S      V300.1, 1                   // M_Alarm_Overflow_BHighR      Q0.4, 1                     // 关阀CMOVW   99, VW2MOVB   2, VB270                    // 故障JMP    6
// 诊断子状态调度LDW=   VW264, 0JMP    1LDW=   VW264, 1JMP    2LDW=   VW264, 2JMP    3LDW=   VW264, 3JMP    4LDW=   VW264, 4JMP    5JMP    6
// ---- 子状态0: 空闲 ----// S0空闲LBL    1JMP    6
// ---- 子状态1: 等待开到位 ----// S1等待开到位LBL    2// T56开到位超时 + T57排水超时(两套独立判据, PT均=VW276)LD     SM0.0TON    T56, VW276                  // PT=VD_Timeout_ValveC(VD54)×10TON    T57, VW276                  // 排水超时: 液位低位未在VD_Timeout_ValveC内到达
// 开到位=ON → 转S2排水中// [已修复 v2.2] 用 V63.2 缓存 EU 结果,避免 R 指令链栈空LD     I8.4EU=      V63.2LD     V63.2MOVW   2, VW264LD     V63.2R      T56, 1LD     V63.2R      T57, 1JMP    6
// 开到位超时 → 报警46LD     T56S      V302.6, 1                   // M_Alarm_ValveC_OpenTimeoutMOVW   99, VW2MOVW   2, VW270JMP    6
// 排水超时(开阀后液位低位仍未到达) → 报警60LD     T57AN     I1.0                        // 确认液位计B低位仍OFFS      V303.0, 1                   // M_Alarm_ValveC_CloseTimeout(排水超时同用码60)MOVW   99, VW2MOVW   2, VW270JMP    6
// ---- 子状态2: 排水中(等待液位低位) ----// S2排水中LBL    3// 液位计B低位=ON → 转S3延时验证LD     I1.0MOVW   3, VW264JMP    6// 液位低位=OFF → 继续排水,无动作
// ---- 子状态3: 延时验证(液位低位须持续ON) ----// S3延时验证LBL    4// I1.0持续ON达VD_Delay_ValveC_Verify → 排水完成,关阀C// 注: I1.0中途OFF时TON输入断开,T101自动清零,液位低位须连续保持LD     I1.0TON    T101, VW284                  // PT=VD_Delay_ValveC_Verify(VD472)×10LD     T101R      Q0.4, 1                     // 关阀CMOVW   4, VW264                    // 转S4等关到位JMP    6// 液位低位丢失 → 回S2排水中(T101已自动复位)LDN    I1.0MOVW   2, VW264JMP    6
// ---- 子状态4: 等待关到位 ----// S4等待关到位LBL    5// T58关到位超时LD     SM0.0TON    T58, VW276                  // PT=VD_Timeout_ValveC×10
// 关到位=ON → 正常完成// [已修复 v2.2] 用 V63.3 缓存条件,避免 R 指令链栈空LD     I8.5=      V63.3LD     V63.3MOVW   0, VW264                    // VW264=0空闲LD     V63.3MOVW   1, VW270                    // Diag_Result_C=1正常完成LD     V63.3R      T58, 1JMP    6
// 关到位超时 → 报警60LD     T58AN     I8.5S      V303.0, 1                   // M_Alarm_ValveC_CloseTimeoutMOVW   99, VW2MOVW   2, VW270                    // Diag_Result_C=2故障(已修正:用MOVW)JMP    6
// 诊断结束LBL    6

// ============================================================// 文件结束// 说明://   1. FC17调用本FC前置VW264=1启动//   2. FC17检查VW270: 0等待, 1正常完成转S5/S7, 2故障//   3. VW276=VD_Timeout_ValveC(VD54)×10转换值//      VW284=VD_Delay_ValveC_Verify(VD472)×10转换值【v10.4新增】//   4. 【v10.4硬件变更】I0.2保留未使用//      V302.5/V302.7/V303.1改为保留位(报警码45/47/61废弃,不再置位)//      T57由"流量开关超时"改制为"排水超时"(液位低位到达超时)//      排水异常=开到位超时(46)或排水/关到位超时(60)//   5. VW270写入统一用MOVW(写完整WORD),确保FC17的AW=VW270判断正确// ============================================================

JMP    6
LBL    1
JMP    6
LBL    2
LD     SM0.0
TON    T56, VW276
TON    T57, VW276
LD     I8.4
EU
=      V63.2
LD     V63.2
MOVW   2, VW264
LD     V63.2
R      T56, 1
LD     V63.2
R      T57, 1
JMP    6
LD     T56
S      V302.6, 1
MOVW   99, VW2
MOVW   2, VW270
JMP    6
LD     T57
AN     I1.0
S      V303.0, 1
MOVW   99, VW2
MOVW   2, VW270
JMP    6
LBL    3
LD     I1.0
MOVW   3, VW264
JMP    6
LBL    4
LD     I1.0
TON    T101, VW284
LD     T101
R      Q0.4, 1
MOVW   4, VW264
JMP    6
LDN    I1.0
MOVW   2, VW264
JMP    6
LBL    5
LD     SM0.0
TON    T58, VW276
LD     I8.5
=      V63.3
LD     V63.3
MOVW   0, VW264
LD     V63.3
MOVW   1, VW270
LD     V63.3
R      T58, 1
JMP    6
LD     T58
AN     I8.5
S      V303.0, 1
MOVW   99, VW2
MOVW   2, VW270
JMP    6
LBL    6
END_SUBROUTINE_BLOCK
SUBROUTINE_BLOCK RhythmCorrection:SBR19
TITLE=// ============================================================
// // 文件: FC40_RhythmCorrection.stl
// // 功能: 双倒计时器周期管理(v2.2 重写,替代原三层纠偏)
// // Story: v2.2 流程重构 (替代 AQEX-8 节奏纠偏)
// // 说明: v2.2 取消原"三层自动纠偏"机制,改为通过 FC40 管理两个交替工作
// //       的 32 位秒计数器(VD248/VD252),严格保证 24h 换水次数硬约束
// // 调用: OB1 每周期调用(在 FC1 状态调度之前)
// // 输出: 触发 S6 排水 / 触发下一轮 S1 / 倒计时到 0 报警 / 双计时器显示值
// // ============================================================
//
// // 符号说明:
// // VD414 : VD_24h_Target           24h 换水目标次数 (HMI 设定)
// // VD426 : VD_Transfer_Margin      周期尾端转移余量 (秒, 默认 30, HMI 设定)
// // VD430 : VD_Prep_Safety_Margin   上缸配液安全余量 (秒, 默认 10, HMI 设定)
// // VD186 : VD_T_cycle              本轮倒计时总时长(秒,内部中间变量)
// // VD248 : VD_TimerA_Elapsed       TimerA 已运行秒数(32 位 REAL)
// // VD252 : VD_TimerB_Elapsed       TimerB 已运行秒数(32 位 REAL)
// // VD256 : VD_TimerA_Display       TimerA 显示值(秒, DINT, HMI 读取)
// // VD244 : VD_TimerB_Display       TimerB 显示值(秒, DINT, HMI 读取)
// // T63   : T_1s_Pulse              1 秒脉冲发生器(100ms 时基,PT=10)
// // V63.4 : M_1s_Pulse              1 秒脉冲 EU 缓存
// // V63.5 : M_S6Trig_Cache          S6触发条件缓存(v2.3, 避免LPS/LPP/ALD栈消耗)
// // V63.6 : M_NextS1Trig_Cache      下一轮S1触发条件缓存(v2.3)
// // V63.7 : M_CycleTimeout_Cache    周期超时报警条件缓存(v2.3)
// // AC2   : 运算中间值(v2.3 NET5 T_cycle-Prep_Needed 阈值)
// // VW2   : 下缸主状态机
// // VW418 : 上缸配液子流程状态
// // VW6   : 当前报警码 (=0 才允许触发)
// // VW400 : 已完成换水次数 (v2.3.2由VW306迁入, 避让手动命令位V306.0~V307.3)
// // VD70  : S1 实测时长 (秒)
// // VD28  : S2 搅拌固定时长 (秒)
// // VD116 : S6 滚动实测时长 (秒,首轮为S4实测值)
// // M16.0 : M_TimerA_Active         当前下缸轮次使用 TimerA 标志
// // M16.1 : M_NextCycleTrigger      触发下一轮 S1 脉冲
// // V303.6: M_Alarm_CycleTimeout    单轮换水周期超时报警
BEGIN
Network 1
//  计算 T_single 和 T_cycle
//  T_single = 86400.0 / VD414          // 单次目标周期(秒)
//  T_cycle = T_single - VD426 - VD430  // 实际倒计时总时长(秒)
LD     SM0.0MOVR   86400.0, VD186/R     VD414, VD186                 // T_single-R     VD426, VD186                 // - Transfer_Margin-R     VD430, VD186                 // - Safety_Margin = T_cycle

// T_cycle <= 0 检查:周期参数过激进,报警并禁止启动LD     SM0.0AR>    VD186, 0.0                   // T_cycle > 0 ?JMP    10                          // 是 → 正常路径// 否 → 参数过激进LD     SM0.0S      V303.6, 1                   // M_Alarm_CycleTimeout=1(强制人工确认)JMP    9                           // → 跳到本FC末尾
LBL    10// 正常路径继续JMP    10
LD     SM0.0
S      V303.6, 1
JMP    9
LBL    10
Network 2
//  1 秒脉冲发生器(100ms 时基,PT=10)
//  [已修复 v2.2] 用 T63 产生 1s 脉冲,驱动 32 位秒计数器,不受 32767 限制
LD     SM0.0R      T63, 1TON    T63, 10LD     T63EU=      V63.4                       // 1 秒脉冲 EU 缓存R      T63, 1
TON    T63, 10
LD     T63
EU
=      V63.4
Network 3
//  双倒计时器累加:本轮进行中,每秒给当前活动计时器 +1
//  【v2.3修复】原门控"仅VW418=1(S1期间)"导致Elapsed只计到S1结束,
//    NET4/NET5的T_cycle比较式永远无法触发;改为"本轮进行中"门控:
//    VW418≠0(上缸子流程进行中) 且 VW2?{0,7,8,99}(非S0/S6/S7/S_ERROR)
//    计时区间为 本轮S6完成→本轮S6触发(排水窗口冻结,与NET4阈值语义对齐)
//  【2026-09-25修复】增加 VW2≠7: S6排水期间冻结计数,消除排水末越界误报
LD     V63.4                       // 1 秒脉冲LDW<>  VW418, 0                    // 上缸子流程进行中(1/2/3/4)AW<>   VW2, 0                      // 非S0AW<>   VW2, 7                      // 【2026-09-25修复】非S6(排水窗口冻结计数,消除越界误报)AW<>   VW2, 8                      // 非S7AW<>   VW2, 99                     // 非S_ERRORA      M16.0                       // TimerA 活动?+R     1.0, VD248                  // TimerA_Elapsed + 1LD     V63.4                       // 1 秒脉冲LDW<>  VW418, 0                    // 上缸子流程进行中AW<>   VW2, 0                      // 非S0AW<>   VW2, 7                      // 【2026-09-25修复】非S6(排水窗口冻结计数)AW<>   VW2, 8                      // 非S7AW<>   VW2, 99                     // 非S_ERRORAN     M16.0                       // TimerB 活动?+R     1.0, VD252                  // TimerB_Elapsed + 1Network 4
//  S6 触发条件
//  【v2.3修复】原实现"Elapsed <= VD116"比较方向与语义相反(且代码注释与指令矛盾),
//    按设计语义改为: 本轮剩余 <= S6_actual ? Elapsed >= T_cycle - VD116
//  S6_actual 统一使用 VD116:首轮为S4实测值(由FC15写入),后续为S6滚动实测值(由FC17写入)
LD     SM0.0LPSA      M16.0                       // 当前 TimerA?MOVR   VD248, AC0                  // AC0 = TimerA_ElapsedLPPLPSAN     M16.0                       // 当前 TimerB?MOVR   VD252, AC0                  // AC0 = TimerB_ElapsedLPPOLD                                // 选择当前活动 ElapsedMOVR   VD186, AC1                  // AC1 = T_cycle-R     VD116, AC1                  // AC1 = T_cycle - S6_actual (S6触发阈值)-R     AC1, AC0                    // AC0 = Elapsed - 阈值AR>=   AC0, 0.0                    // Elapsed >= T_cycle - S6_actual ?AW=    VW2, 6                      // 当前在 S5AW=    VW6, 0                      // 无报警=      V63.5                       // 缓存S6触发条件(避免LPS/LPP/ALD栈消耗丢弃门控)LD     V63.5MOVW   7, VW2                      // 转 S6 排水LD     V63.5S      M10.7, 1                    // 【v2.3修复】置S6首次进入脉冲(原FC16已删除置位,FC17无源可取)AW=    VW2, 6
AW=    VW6, 0
=      V63.5
LD     V63.5
MOVW   7, VW2
LD     V63.5
S      M10.7, 1
Network 5
//  下一轮 S1 触发条件
//  【v2.3修复】原实现"Elapsed >= Prep_Needed"漏T_cycle项,且要求VW418=0(死条件);
//    按设计语义改为: 本轮剩余 <= Prep_Needed ? Elapsed >= T_cycle - Prep_Needed,
//    门控改为 VW418=4(上缸已转移,可启动下一轮配液)
//  Prep_Needed = VD70 + VD28 + VD430 (S1 实测 + S2 固定 + 上缸安全余量)
LD     SM0.0LPSA      M16.0                       // 当前 TimerA?MOVR   VD248, AC0                  // AC0 = TimerA_ElapsedLPPLPSAN     M16.0                       // 当前 TimerB?MOVR   VD252, AC0                  // AC0 = TimerB_ElapsedLPPOLD                                // 选择当前活动 ElapsedMOVR   VD70, AC1                   // AC1 = S1_Actual+R     VD28, AC1                   // + S2 固定+R     VD430, AC1                  // + 安全余量 = Prep_NeededMOVR   VD186, AC2                  // AC2 = T_cycle-R     AC1, AC2                    // AC2 = T_cycle - Prep_Needed (下一轮S1触发阈值)-R     AC2, AC0                    // AC0 = Elapsed - 阈值AR>=   AC0, 0.0                    // Elapsed >= T_cycle - Prep_Needed ?AW=    VW418, 4                    // 【v2.3修复】上缸已转移(原VW418=0为死状态)AW=    VW6, 0                      // 无报警=      V63.6                       // 缓存触发条件LD     V63.6S      M16.1, 1                    // 触发下一轮 S1 脉冲(由OB1消费: VW418 4→1)AR>=   AC0, 0.0
AW=    VW418, 4
AW=    VW6, 0
=      V63.6
LD     V63.6
S      M16.1, 1
Network 6
//  倒计时到 0 报警 (V303.6)
//  报警语义: "错过S6触发窗口"才报 —— Elapsed >= T_cycle 且 NET4 本扫描未触发 S6
//  【2026-09-25修复】原门控仅"不在S7",导致:
//    (a) VD116=0(首轮)时 NET4/NET6 同阈值,NET4先置VW2=7,NET6同扫描误报;
//    (b) S6排水期间 NET3 继续累加,排水末 Elapsed 必然越界,每轮末必报
//    修复: AN V63.5(S6触发缓存) + 排除 VW2=7(S6排水窗口,计数已冻结)
//  【v2.3修复】原LPS/LPP/ALD结构会丢弃门控,改用V位缓存
LD     SM0.0LPSA      M16.0                       // 当前 TimerA?MOVR   VD248, AC0                  // AC0 = TimerA_ElapsedLPPLPSAN     M16.0                       // 当前 TimerB?MOVR   VD252, AC0                  // AC0 = TimerB_ElapsedLPPOLD                                // 选择当前活动 Elapsed-R     VD186, AC0                  // AC0 = Elapsed - T_cycleAR>=   AC0, 0.0                    // Elapsed >= T_cycle ?AN     V63.5                       // 【2026-09-25】NET4未在本扫描触发S6(错过窗口才报)AW<>   VW2, 7                      // 【2026-09-25】不在S6排水窗口(计数冻结,Elapsed不再增长)AW<>   VW2, 8                      // 不在 S7=      V63.7                       // 缓存报警条件LD     V63.7S      V303.6, 1                   // 单轮换水周期超时报警AN     V63.5
AW<>   VW2, 7
AW<>   VW2, 8
=      V63.7
LD     V63.7
S      V303.6, 1
Network 7
//  双倒计时器显示值写入 (HMI 读取)
//  [已修复 v2.2] VD256/VD244 直接显示 Elapsed 秒数(DINT)
LD     M16.0                       // 当前使用 TimerA?
ROUND  VD248, VD256                // VD_TimerA_Display = TimerA_Elapsed (秒)LDN    M16.0                       // 当前使用 TimerB?ROUND  VD252, VD244                // VD_TimerB_Display = TimerB_Elapsed (秒)

LBL    9// 本FC结束// 返回 OB1 (OB1 在调度 FC1 之前调用本FC,保证 M16.1 下一轮 S1 触发脉冲及时响应)

// ============================================================// 文件结束// ============================================================// 说明://   1. 调用时机: OB1 在 FC22(RTC Sync) 之后、FC1(状态调度) 之前调用//   2. 计数器清零: FC11 在 S1 首次进入时清零【非活动】计数器//      (S1启动于本轮中段,活动计数器属于本轮,不能清;计时区间为 S6完成→S6触发)//   3. 计时器切换: S6 完成后由 FC17 切 M16.0 = NOT M16.0(全程序唯一切换点)//   4. 报警 V303.6: 不受 V200.0 模式影响,必须 V0.3 人工确认;//      置位条件为"错过S6触发窗口"(NET4未触发且Elapsed>=T_cycle且不在S6/S7);//      复位由 FC3 NETWORK 4 (V0.3上升沿) 执行: 清V303.6 + 清零VD248/VD252(本轮重新计时),//      FC3A 公共复位不含此位(2026-09-25补漏); 不清计时器则确认后同扫描被NET6重报(死锁)//   5. T_cycle <= 0: 直接报警并跳过本周期其他计算(跳到 LBL 9)//   6. 显示值 VD256/VD244: 真空闲区(原 VD442/VD446 与 VD440/444 字节重叠已迁移)// ============================================================

LBL    9
END_SUBROUTINE_BLOCK
SUBROUTINE_BLOCK MBUS_CTRL:SBR20
TITLE=This code is property of Siemens Industry, Inc.
VAR_INPUT
Mode:BOOL;	//  1 = Modbus, 0 = PPI (stop Modbus)
Baud:DWORD;	//  1200, 2400 ... 115200
Parity:BYTE;	//  0 = none, 1 = odd, 2 = even
Port:BYTE;	// 0 or 1
Timeout:INT;	//  slave response timeout in milliseconds
END_VAR
VAR_OUTPUT
Done:BOOL;	//  Done flag (always set)
Error:BYTE;	//  Error status
END_VAR
VAR
AC0save:DWORD;
AC1save:DWORD;
AC2save:DWORD;
AC3save:DWORD;
END_VAR
BEGIN
Network 1 // 此 POU 针对编辑和查看设置了密码保护.

END_SUBROUTINE_BLOCK
SUBROUTINE_BLOCK MBUS_MSG:SBR21
TITLE=This code is property of Siemens Industry, Inc.
VAR_INPUT
First:BOOL;	// New message (Set to a 1 for only one scan for a new request)
Slave:BYTE;	// Slave address (0 - 247)
RW:BYTE;	// Read = 0, Write = 1
Addr:DWORD;	// Modbus addr (ie 40001)
Count:INT;	// Number of elements (1- 120 words or 1 to 1920 bits)
DataPtr:DWORD;	// Pointer to data (ie &VB100)
END_VAR
VAR_OUTPUT
Done:BOOL;	// Done flag (0 = busy, 1 = done)
Error:BYTE;	// Error (0 = no error)
END_VAR
VAR
AC0save:DWORD;
AC1save:DWORD;
AC2save:DWORD;
END_VAR
BEGIN
Network 1 // 此 POU 针对编辑和查看设置了密码保护.

END_SUBROUTINE_BLOCK
SUBROUTINE_BLOCK MBUSM1:SBR22
TITLE=This code is property of Siemens Industry, Inc.
VAR_OUTPUT
crc:WORD;
END_VAR
VAR
count:INT;
ptr:DWORD;
END_VAR
BEGIN
Network 1 // 此 POU 针对编辑和查看设置了密码保护.

END_SUBROUTINE_BLOCK
SUBROUTINE_BLOCK ManualSyringePump:SBR23
TITLE=
BEGIN
Network 1
//  孤儿态自恢复
//  [已修复 v2.2] 用 V62.2 缓存条件,避免 R 指令链栈空
LDW<>  VW390, 0
AW<>   VW390, 30
AN     M11.6
AN     M11.7
AN     M12.0
AN     M13.5
AN     M13.6
=      V62.2
LD     V62.2
MOVW   0, VW390
LD     V62.2
R      M13.7, 1


// 启动命令检测 - 仅空闲态(VW390=0)响应
// [已修复 v2.2] 用 V62.3 缓存 EU 结果,避免 S/R 指令链栈空
LD     SM0.0
A      V307.2
EU
AW=    VW390, 0
=      V62.3
LD     V62.3
MOVR   0.0, VD392
LD     V62.3
MOVR   VD452, VD396
LD     V62.3
R      M13.7, 1
LD     V62.3
R      M13.5, 1
LD     V62.3
R      M13.6, 1
LD     V62.3
R      M12.0, 1
LD     V62.3
R      M11.6, 1
LD     V62.3
R      M11.7, 1
LD     V62.3
MOVW   1, VW390
LD     V62.3
R      V307.2, 1


// 停止命令检测 - 非空闲态响应
// [已修复 v2.2] 用 V62.4 缓存 EU 结果,避免 S/R 指令链栈空
LD     SM0.0
A      V307.3
EU
AW<>   VW390, 0
=      V62.4
LD     V62.4
S      M13.7, 1
LD     V62.4
R      V307.3, 1


// 全局错误检测
// [已修复 v2.2] 用 V62.5 缓存全局错误条件,避免 R 指令链栈空
LDW=   VW390, 1
OW=    VW390, 2
OW=    VW390, 3
LD     V303.4
LD     SM0.0
AW>=   VW4, 4
OLD
ALD
=      V62.5
LD     V62.5
MOVW   99, VW390
LD     V62.5
R      M13.5, 1
LD     V62.5
R      M13.6, 1
LD     V62.5
R      M13.7, 1
LD     V62.5
R      M12.0, 1
LD     V62.5
R      M11.6, 1
LD     V62.5
R      M11.7, 1


// 子状态1-1 - 计算本次抽液步数
LD     SM0.0
AW=    VW390, 1
AN     M13.5
AN     M11.6
AN     M11.7
AN     M12.0
MOVR   VD396, VD102
/R     VD350, VD102
AR>=   VD102, 6000.0
JMP    10
ROUND  VD102, AC0
MOVR   AC0, VD102
JMP    11
LBL    10
MOVR   6000.0, VD102
LBL    11


// 子状态1-2 - 检查步数并下发抽液指令(40006)
LD     SM0.0
AW=    VW390, 1
AN     M13.5
AN     M11.6
AN     M11.7
AN     M12.0
AW=    VW4, 0
=      V60.4
LD     V60.4
ROUND  VD102, AC0
AR>    AC0, 0.0
JMP    12
// [已修复 v2.2] 复用 V60.4 缓存条件,补齐 R/S 链前面的 LD
LD     V60.4
R      M12.0, 1
LD     V60.4
R      M11.6, 1
LD     V60.4
R      M11.7, 1
LD     V60.4
MOVW   3, VW390
JMP    13
LBL    12
MOVW   AC0, VW204
MOVW   AC0, VW230
MOVD   16#9C46, VD232
LD     V60.4
S      M11.6, 1
LD     V60.4
S      M13.5, 1
LBL    13


// 子状态1-3 - 抽液写失败处理
// [已修复 v2.2] 用 V64.0 缓存条件,避免 S/R 链栈空
LD     M12.0
AW=    VW390, 1
A      V303.4
=      V64.0
LD     V64.0
MOVW   99, VW390
LD     V64.0
R      M13.5, 1
LD     V64.0
R      M13.7, 1
LD     V64.0
R      M12.0, 1
LD     V64.0
R      M11.6, 1
LD     V64.0
R      M11.7, 1


// 子状态1-3 - 抽液写成功处理
// [已修复 v2.2] 用 V64.1 缓存条件,避免 S/R 链栈空
LD     M12.0
AW=    VW390, 1
AN     V303.4
=      V64.1
LD     V64.1
R      M12.0, 1
LD     V64.1
R      M11.6, 1


// 子状态1-4 - 等待抽液执行完成
// [已修复 v2.2] 用 V65.4 缓存条件,避免 R 指令链栈空
LD     M13.5
AW=    VW390, 1
AW=    VW4, 0
AN     M11.6
AN     M11.7
AN     M12.0
=      V65.4
LD     V65.4
R      M13.5, 1
LD     V65.4
MOVW   2, VW390


// 子状态2-1 - 下发排液指令(40007)
// [已修复 v2.2] 用 V65.3 缓存条件,避免 S 指令链栈空
LD     SM0.0
AW=    VW390, 2
AN     M13.6
AN     M11.6
AN     M11.7
AN     M12.0
AW=    VW4, 0
=      V65.3
LD     V65.3
ROUND  VD102, AC0
MOVW   AC0, VW230
MOVW   AC0, VW206
MOVD   16#9C47, VD232
LD     V65.3
S      M11.6, 1
LD     V65.3
S      M13.6, 1


// 子状态2-2 - 排液写失败处理
// [已修复 v2.2] 用 V64.2 缓存条件,避免 S/R 链栈空
LD     M12.0
AW=    VW390, 2
A      V303.4
=      V64.2
LD     V64.2
MOVW   99, VW390
LD     V64.2
R      M13.6, 1
LD     V64.2
R      M13.7, 1
LD     V64.2
R      M12.0, 1
LD     V64.2
R      M11.6, 1
LD     V64.2
R      M11.7, 1


// 子状态2-2 - 排液写成功处理
// [已修复 v2.2] 用 V64.3 缓存条件,避免 S/R 链栈空
LD     M12.0
AW=    VW390, 2
AN     V303.4
=      V64.3
LD     V64.3
R      M12.0, 1
LD     V64.3
R      M11.6, 1


// 子状态2-3 - 等待排液执行完成,累加本循环体积
// [已修复 v2.2] 用 V64.4 缓存条件,避免 S/R 链栈空
LD     M13.6
AW=    VW390, 2
AW=    VW4, 0
AN     M11.6
AN     M11.7
AN     M12.0
=      V64.4
LD     V64.4
MOVR   VD102, AC0
LD     V64.4
*R     VD350, AC0
LD     V64.4
+R     AC0, VD392
LD     V64.4
-R     AC0, VD396
LD     V64.4
R      M13.6, 1


// 子状态2-4 - 判断分支: 停止请求 → 回零
// [已修复 v2.2] 用 V64.5 缓存条件,避免 S/R 链栈空
LD     SM0.0
AW=    VW390, 2
AN     M13.6
A      M13.7
=      V64.5
LD     V64.5
R      M12.0, 1
LD     V64.5
R      M11.6, 1
LD     V64.5
R      M11.7, 1
LD     V64.5
MOVW   3, VW390


// 子状态2-4 - 判断分支: 单次模式 → 回零
// [已修复 v2.2] 用 V64.6 缓存条件,避免 S/R 链栈空
LD     SM0.0
AW=    VW390, 2
AN     M13.6
AW=    VW388, 0
=      V64.6
LD     V64.6
R      M12.0, 1
LD     V64.6
R      M11.6, 1
LD     V64.6
R      M11.7, 1
LD     V64.6
MOVW   3, VW390


// 子状态2-4 - 判断分支: 循环模式且累计>=目标 → 回零
// [已修复 v2.2] 用 V64.7 缓存条件,避免 S/R 链栈空
LD     SM0.0
AW=    VW390, 2
AN     M13.6
AW=    VW388, 1
AR>=   VD392, VD452
=      V64.7
LD     V64.7
R      M12.0, 1
LD     V64.7
R      M11.6, 1
LD     V64.7
R      M11.7, 1
LD     V64.7
MOVW   3, VW390


// 子状态2-4 - 判断分支: 循环模式且未完成 → 返回子状态1
// [已修复 v2.2] 用 V65.0 缓存条件,避免 S/R 链栈空
LD     SM0.0
AW=    VW390, 2
AN     M13.6
AW=    VW388, 1
AR<    VD392, VD452
=      V65.0
LD     V65.0
R      M12.0, 1
LD     V65.0
R      M11.6, 1
LD     V65.0
R      M11.7, 1
LD     V65.0
MOVW   1, VW390


// 子状态3-1 - 下发回零(复位)指令 40003=1
LD     SM0.0
LDW=   VW390, 3
OW=    VW390, 30
AN     M11.6
AN     M11.7
AN     M12.0
AW=    VW4, 0
AW=    VW510, 0
O      T104
MOVW   1, VW230
MOVD   16#9C43, VD232
S      M11.6, 1
MOVW   30, VW390


// T104冷却定时器
LD     M12.0
AW=    VW390, 30
AW>    VW510, 0
TON    T104, 50


// 子状态3-2 - 回零写失败处理
// [已修复 v2.2] 用 V65.1 缓存条件,避免 S/R 链栈空
LD     M12.0
AW=    VW390, 30
A      V303.4
=      V65.1
LD     V65.1
MOVW   99, VW390
LD     V65.1
R      M13.7, 1
LD     V65.1
R      M12.0, 1
LD     V65.1
R      M11.6, 1
LD     V65.1
R      M11.7, 1
LD     V65.1
R      T104, 1


// 子状态3-2 - 回零写成功处理
// [已修复 v2.2] 用 V65.2 缓存条件,避免 S/R 链栈空
LD     M12.0
AW=    VW390, 30
AN     V303.4
=      V65.2
LD     V65.2
R      M12.0, 1
LD     V65.2
R      M13.5, 1
LD     V65.2
R      M13.6, 1
LD     V65.2
R      M13.7, 1
LD     V65.2
R      M11.6, 1
LD     V65.2
R      M11.7, 1
LD     V65.2
R      T104, 1
LD     V65.2
MOVW   4, VW390

END_SUBROUTINE_BLOCK
SUBROUTINE_BLOCK RTC_Sync:SBR24
TITLE=// ============================================================
// // 文件: FC22_RTC_Sync.stl
// // 功能: RTC时间同步处理
// // Story: AQEX-51 PLC长时间停机后HMI校时
// // 说明:
// //   1. HMI通过McgsPro将当前时间(BCD格式)写入VB900~VB905
// //   2. HMI置位V0.6(CMD_RTC_Sync)
// //   3. 本FC检测V0.6上升沿，调用TODW将VB900~VB907写入PLC RTC
// //   4. 写入成功后复位V303.7(M_Need_RTC_Sync)和V0.6
// //   5. 若V303.7=1持续5分钟(300秒)未同步，置V303.5并转S_ERROR
// // ============================================================
//
// // 符号说明:
// // V0.6  : CMD_RTC_Sync     HMI校时命令(上升沿触发)
// // V303.5: M_Alarm_RTC_Lost RTC时钟丢失报警(超时未同步后置位)
// // V303.7: M_Need_RTC_Sync  请求HMI同步PLC时间
// // VB900~VB907: RTC时间缓冲区(BCD格式)
// // T59   : 校时超时定时器(100ms时基,5分钟=3000×100ms)子程序注释
BEGIN
Network 1
//  HMI校时命令上升沿检测
//  检测V0.6上升沿 -> 跳到LBL1执行TODW写入RTC
LD     V0.6
EU
JMP    1

// 超时保护: V303.7=1时启动5分钟超时定时器
LD     V303.7
TON    T59, 3000
LD     T59
EU
S      V303.5, 1
MOVW   99, VW2
JMP    2

// 正常路径: 无校时命令且未超时，直接结束
LD     SM0.0
JMP    2

// ============================================================
// LBL1: 执行TODW写入RTC
// ============================================================
LBL    1
LD     SM0.0
MOVB   0, VB906
MOVB   0, VB907
TODW   VB900
R      V303.7, 1
R      V0.6, 1

// ============================================================
// LBL2: 结束
// ============================================================
LBL    2
END_SUBROUTINE_BLOCK
SUBROUTINE_BLOCK ColdStart:SBR25
TITLE=// ============================================================
// // 文件: SBR25_ColdStart.stl
// // 功能: 冷启动路径 — 出厂硬编码 + 用户默认覆盖 + TODR + 安全初始化
// // 调用: 由 FC0_SysInit 在 M16.4=0 (冷启动) 时 CALL
// // 返回: SBR 自然结束回到 FC0,FC0 继续执行 LBL 2 (S M16.4,1)
// // 【v2.2迁移 2026-09-15】M_InitDone 从 V304.0 迁至 M16.4
// // LBL 分配: 8/9/10(用户默认覆盖)、88/89(RTC异常处理)
// // 说明: 拆分自原单一 FC0,内部无跨 SBR JMP/LBL 依赖
// // ★ 重要: S7-200 SMART STL 的 JMP/LBL 必须在同一 NETWORK 内,
// //   因此本 SBR 只保留一个 NETWORK,所有 JMP/LBL 全部在此 NETWORK 中
// // ============================================================
//
BEGIN
Network 1
//  冷启动完整路径(单一NETWORK):
//    1) 出厂硬编码
//    2) 用户默认覆盖(LBL 8/9/10)
//    3) TODR读RTC + 合法性检查(LBL 88/89)
//    4) 安全初始化,SBR 自然结束返回 FC0
//  注射泵单步分辨率(25ml注射器标准6000步模式)
MOVR   4.1667, VD350               // VD_StepResolution

// 6.2 时间周期参数
// 【v2.2 修订 2026-09-15】取消 VD_CycleSetpoint (改用 VD414 24h 目标次数)
//                       取消 VD_PreMixTime_MinSafe / VD_RestTime / VD_RestTime_Min
//                       取消 VD_CycleExtend_Max / VD_T_Default (三层纠偏已删除)
MOVR   10080.0, VD24      // VD_ExperimentTarget 实验总时长(min,默认7天)
MOVR   1800.0, VD28       // VD_PreMixTime S2搅拌固定时长(s,默认30min,v2.2 严格不可压缩)
MOVR   6.0, VD414         // 【v2.2新增】VD_24h_Target 24h换水目标次数(默认6)
MOVR   180.0, VD426       // 【v2.2新增】VD_Transfer_Margin 周期尾端转移余量(s,默认3min)
MOVR   180.0, VD430       // 【v2.2新增】VD_Prep_Safety_Margin 上缸配液安全余量(s,默认3min)

// 6.2.1 工艺目标参数
MOVR   10.0, VD316        // 目标进水量(L,默认10L)
MOVR   5000.0, VD584      // VD_Vol_Target 默认加药量(μL,默认5mL)

// 6.3 超时保护参数
MOVR   60.0, VD358        // VD_Timeout_ValveA 阀A开/关到位超时(s)
MOVR   60.0, VD362        // VD_Timeout_ValveB 阀B开/关到位超时(s)
MOVR   60.0, VD54         // VD_Timeout_ValveC 阀C开/关到位超时(s)
MOVR   60.0, VD66                  // VD_Delay_ValveA_Verify 阀A关后延时验证(s)
MOVR   5.0, VD472                  // 【v10.4新增,2026-09-24由VD60迁来】VD_Delay_ValveC_Verify 阀C液位B低位延时验证(s)
MOVW   1800, VW288        // 【v2.3.2新增】VW_S4_Transfer_PT S4转移计时T49的PT(100ms单位,1800=180s)
                          //   PLC侧无运行时写入方(FC15只读用),此处给冷启动初值,HMI参数页可改

// 7.4 其他超时阈值
MOVR   1800.0, VD448      // VD_S4WaitTimeout S4等待超时阈值(s)
MOVR   10000.0, VD452     // VD_ManualDose_Target 手动总加药量(μL,默认10mL)
MOVW   0, VW388           // VW_ManualDose_Mode 手动模式(0=单次,1=循环)

// ===== 用户默认参数覆盖 =====
LDB=   VB456, 1              // VB456 == 1 (用户默认有效)?
JMP    8                     // 是 → 跳 LBL 8 执行用户默认覆盖
LD     SM0.0                 // 强制 C0=1
JMP    9                     // 无条件跳 LBL 9 (跳过覆盖)

LBL    8                     // ====== 用户默认覆盖区 ======
// 【v2.2 修订 2026-09-15】删除 VD468/VD472/VD476/VD480/VD496/VD508 等已废弃变量覆盖
// 【v2.2.1 修订 2026-09-17】VD468/VD476/VD480 重新分配为 v2.2 时间参数 (VD414/426/430)
//                         的用户默认镜像 (经字节级 + 字级 + 双字级 + 间接访问四维核实,
//                         VW236 (bytes 472-473) / VW252 (bytes 504-505) 不与新地址重叠);
//                         VD496/VD508 仍保留为空 (待未来扩展); VD472 已于 2026-09-24 分配给 VD_Delay_ValveC_Verify
MOVR   VD460, VD24           // VD_ExperimentTarget
MOVR   VD464, VD28           // VD_PreMixTime (S2搅拌固定时长)
MOVR   VD484, VD54           // VD_Timeout_ValveC
MOVR   VD488, VD66           // VD_Delay_ValveA_Verify
// 【2026-09-24决策】恢复无条件覆盖：出厂默认防0的责任在HMI侧——HMI首次运行/参数页打开时
//   须把出厂默认值写入整个镜像区(VD460~VD536)并置VB456=1，PLC不做非0门控
MOVR   VD492, VD472          // 【v3.1新增,2026-09-24由VD60迁来】UD_VD60_DelayC → VD_Delay_ValveC_Verify 排液完成验证延时
                             //   (原VD60因与V60.x~V63.x EU缓存位区重叠而废弃; VD472经字节/字/双字/位四维核实无占用)
MOVR   VD500, VD316          // VD_TargetInletVolume
MOVR   VD504, VD350          // VD_StepResolution
MOVR   VD512, VD358          // VD_Timeout_ValveA
MOVR   VD516, VD362          // VD_Timeout_ValveB
MOVR   VD520, VD584          // VD_Vol_Target
MOVR   VD524, VD448          // VD_S4WaitTimeout
MOVR   VD528, VD452          // VD_ManualDose_Target
MOVR   VD468, VD414          // UD_VD414_24h_Target         (v2.2 新增, 24h 换水目标次数, 默认6)
MOVR   VD476, VD426          // UD_VD426_Transfer_Margin    (v2.2 新增, 周期尾端转移余量, 默认180s)
MOVR   VD480, VD430          // UD_VD430_Safety_Margin      (v2.2 新增, 上缸配液安全余量, 默认180s)

// WORD: VW388 ManualDose_Mode
MOVB   VB532, VB388           // 复制低字节
MOVB   0, VB389               // 高字节清零

// BIT: V200.0 AlarmAckMode
LDB=   VB536, 1
JMP    10                     // VB536 == 1 → 跳去 S V200.0
R      V200.0, 1              // VB536 != 1 → 清 V200.0
LD     SM0.0
JMP    9                      // 无条件跳汇合点
LBL    10
S      V200.0, 1              // VB536 == 1 → 置 V200.0

// LBL 9 汇合 → TODR读RTC + 合法性检查 (LBL 88/89)
LBL    9                     // ====== 覆盖后汇合点 ======

// 实验总换水次数目标计算(v2.2新增)
// VW8 = VD414(24h换水目标次数) × VD24(实验总时长min) / 1440
LD     SM0.0
MOVR   VD414, AC0
*R     VD24, AC0
/R     1440.0, AC0
ROUND  AC0, AC0
DTI    AC0, VW8

// ★ 2026-09-13: 冷启动也要读PLC内部RTC到VB900~VB907
LD     SM0.1
TODR   VB900

// RTC自身合法性检查(RTC字段越界+年份归零→请求校时)
// ★ 2026-09-13新增: 年份合理性检查(超级电容归零→VB900=00→2000年)
LDB<   VB900, 20          // 年<20(2020年前) → RTC不可信
JMP    88
LDB>   VB901, 12          // 月>12
JMP    88
LDB<   VB901, 1           // 月<1
JMP    88
LDB>   VB902, 31          // 日>31
JMP    88
LDB<   VB902, 1           // 日<1
JMP    88
LDB>   VB903, 23          // 时>23
JMP    88
LDB>   VB904, 59          // 分>59
JMP    88
LDB>   VB905, 59          // 秒>59
JMP    88
LD     SM0.0              // RTC正常 → 跳过异常处理
JMP    89

LBL    88                 // 冷启动RTC异常
LD     SM0.1
S      V303.7, 1          // 请求HMI校时

LBL    89                 // 汇合点

// 状态机初始化为S0
MOVW   0, VW2             // VW2=0(S0)
// 冷启动也清阀门诊断子状态和计时器
FILL   0, VW260, 8        // 清 VB260~VB275
R      T50, 6             // 清 T50~T55
R      V1.6, 1            // 上缸=空
R      V1.7, 1            // 下缸=空

// 复位所有DO输出(安全状态)
MOVB   0, QB0             // Q0.0~Q0.7=0
MOVB   0, QB8             // Q8.0~Q8.7=0

// 清除急停锁存
R      V300.4, 1          // M_EStop_Latch=0

// 清除报警字和报警码
// 【2026-09-29修复】FILL第三操作数是字数非字节数: 原"4"实际清VW300/302/304/306(VB300~307),
//   每次冷启动把上缸子流程状态VW418连带清0(交叉引用实证)。改为2字=VB300~303, 与注释一致
FILL   0, VW300, 2        // VW300~VW301(=VB300~VB303)清零
MOVW   0, VW6             // VW6=0(无报警)

// 清除FC3内部继电器
R      M11.1, 1           // M_Sound_Latched=0
R      M11.2, 1           // M_PrevAlarm=0

// 冷启动必须清 VB0,防止 V0.x 命令位断电保持后卡1
MOVB   0, VB0             // V0.0~V0.7 全部清0
R      V1.0, 6            // V1.0~V1.5=0

// 本次实验累计流量清零
MOVR   0.0, VD406         // VD_ExpTotal_Flow=0(L) (原VD364,2026-09-29迁移:与VD366重叠2字节;VD402槽被VW402(T38_PT)占)

// 本次实验累计加药量清零
MOVR   0.0, VD440         // VD_Dosed_Volume_Total=0(μL)

// S4等待时长清零
MOVR   0.0, VD444

// S3剩余待加药量清零
MOVR   0.0, VD372         // VD_Remaining_Vol=0(μL)

// 清下缸满计时器+预规划标志
MOVR   0.0, VD178         // VD_S5_Elapsed=0
R      M10.7, 1
R      M10.2, 1           // 【2026-09-29新增】清S1首次进入标志(v2.2重构丢失置位点后的防御性清理)

// 初始化Modbus轮询计数器与状态
FILL   0, VW290, 4        // VW290~VW296 清零
R      M10.0, 6
LD     SM0.1
R      T103, 1
S      M15.0, 1           // 首次扫描启动任务0
R      M15.1, 1
R      M15.2, 1
R      V60.0, 8           // [已修复 v2.2] 扩展到 V60.7,覆盖 FC4 任务切换新增中间继电器
R      M11.0, 1
R      M11.6, 3                    // M11.6, M11.7, M12.0 (连续3位)
R      M16.5, 1                    // 清注射泵在线标志(v2.2迁移自V304.1)
R      M16.6, 1                    // 清流量计在线标志(v2.2迁移自V304.2)
R      M12.1, 2                    // M12.1, M12.2 (连续2位)
R      M13.0, 5                    // 清手动控制锁存
R      M13.5, 3           // 清手动注射泵标志
MOVW   0, VW390           // 手动注射泵子状态=0
MOVR   0.0, VD392
MOVR   0.0, VD396

// 清错误码/写目标地址
FILL   0, VW378, 3        // 清 VB378~VB383 (6字节合并)
MOVR   0.0, VD374
MOVW   0, VW226
MOVD   0, VD232
MOVW   0, VW230
// ★ 冗余段已删除: 不再重复清 VD232/VW230/M11.6 (上面已清)
// ★ 冗余段已删除: VD414/VD426/VD430 已在出厂硬编码段设置

// 【v2.2 新增】冷启动时初始化上缸子流程 + 双倒计时器显示值清零
MOVW   0, VW418                     // 上缸配液子流程状态清零(防御性)
MOVW   0, VW400                     // 换水计数清零 【v2.3.2迁移: 原VW306与手动命令位V306.0~V307.3重叠】
R      M16.0, 4                     // M16.0~M16.3 连续清零
R      T63, 1                       // [已修复 v2.2] 清 1s 脉冲定时器
MOVR   0.0, VD248                   // TimerA_Elapsed 清零
MOVR   0.0, VD252                   // TimerB_Elapsed 清零
MOVR   0.0, VD256                   // TimerA 显示值清零
MOVR   0.0, VD244                   // TimerB 显示值清零

MOVW   2, VW198           // 步骤=2(冷启动完成)
// SBR 自然结束,返回到 FC0 的 LBL 2 (S M16.4,1)


// ============================================================
// 文件结束
// ============================================================

END_SUBROUTINE_BLOCK
SUBROUTINE_BLOCK WarmRecovery:SBR26
TITLE=// ============================================================
// // 文件: SBR26_WarmRecovery.stl
// // 功能: 断电恢复路径 — RTC检测 + BCD转秒 + 状态机恢复
// // 调用: 由 FC0_SysInit 在 M16.4=1 (断电恢复) 时 CALL
// // 返回: SBR 自然结束回到 FC0,FC0 继续执行 LBL 2 (S M16.4,1)
// // 【v2.2迁移 2026-09-15】M_InitDone 从 V304.0 迁至 M16.4
// // LBL 分配: 1(入口)、3(RTC正常)、4(RTC异常)、5(状态恢复)、6(保持)、7(S_ERROR)、10(S_ERROR回S0清理,兼S5残留清理落点)
// // 【2026-09-29修复】S5保持加前提(V1.7=1或VW418≠0),无前提时跳LBL10复用清理段回S0(不为S5单写副本,省程序存储器)
// // 说明: 拆分自原单一 FC0,原来的 JMP 2(跳FC0完成点) 全部改为 SBR 自然结束
// //   注意: 断电恢复路径不清报警字,VW300~303/VW6/V300.x 由 FC3/FC19 按确认流程处理
// // ★ 重要: S7-200 SMART STL 的 JMP/LBL 必须在同一 NETWORK 内,
// //   因此本 SBR 只保留一个 NETWORK,所有 JMP/LBL 全部在此 NETWORK 中
// // ============================================================
BEGIN
Network 1
//  断电恢复完整路径(单一NETWORK):
//    1) TODR读RTC + 合法性检查 + DT10比较(LBL 1/3/4)
//    2) BCD转秒 + VD_S5_Elapsed重算(LBL 3/5)
//    3) 状态机恢复策略(LBL 5/6/7),SBR 自然结束返回 FC0
//  LBL 1: 入口 (FC0 通过 CALL WarmRecovery 进入,从 LBL 1 开始执行)

// 【2026-09-24新增】暖启动参数NaN自愈: 新PLC未清除V区/异常写入可能使REAL为NaN,//   暖启动不执行SBR25出厂默认段, NaN会永久残留, 并导致HMI参数页"应用设置"把NaN缓冲//   往返写回(表现为改了参数值不变)。利用IEEE754规则"NaN与自身不等"检测, 命中即恢复出厂默认LD     SM0.0AR<>   VD472, VD472                  // VD472是NaN ? (NaN<>NaN恒真)MOVR   5.0, VD472                    // 是 → 恢复出厂默认5.0LD     SM0.1TODR VB900                // 读RTC到VB900~VB907(BCD)
// RTC自身合法性检查(RTC字段越界→请求校时)LDB>   VB901, 12          // 月>12JMP    4LDB<   VB901, 1           // 月<1JMP    4LDB>   VB902, 31          // 日>31JMP    4LDB<   VB902, 1           // 日<1JMP    4LDB>   VB903, 23          // 时>23JMP    4LDB>   VB904, 59          // 分>59JMP    4LDB>   VB905, 59          // 秒>59JMP    4
// RTC丢失检测: 比较RTC与DT10(VB10~VB17)LDB=   VB10, 0            // DT10未写入 → 跳过检测JMP    3
// DT10数据合法性检查（防止历史垃圾数据误触发RTC丢失）LDB<   VB11, 1            // 月<1JMP    4LDB>   VB11, 12           // 月>12JMP    4LDB<   VB12, 1            // 日<1JMP    4LDB>   VB12, 31           // 日>31JMP    4LDB>   VB13, 23           // 时>23JMP    4LDB>   VB14, 59           // 分>59JMP    4LDB>   VB15, 59           // 秒>59JMP    4
// 逐字段BCD比较(年→月→日→时→分→秒)LDB<   VB900, VB10        // RTC年 < DT10年 → RTC丢失JMP    4LDB>   VB900, VB10        // RTC年 > DT10年 → 正常JMP    3LDB<   VB901, VB11        // 比月JMP    4LDB>   VB901, VB11JMP    3LDB<   VB902, VB12        // 比日JMP    4LDB>   VB902, VB12JMP    3LDB<   VB903, VB13        // 比时JMP    4LDB>   VB903, VB13JMP    3LDB<   VB904, VB14        // 比分JMP    4LDB>   VB904, VB14JMP    3LDB<   VB905, VB15        // 比秒JMP    4LD     SM0.0              // 全部>= → RTC正常JMP    3
// RTC异常/丢失 → 请求HMI校时LBL    4LD     SM0.1S      V303.7, 1          // M_Need_RTC_SyncMOVR   0.0, VD178         // VD_S5_Elapsed=0(无法重算)MOVW   3, VW198           // 步骤=3(RTC需校时)JMP    5                  // → 状态恢复
// RTC正常，继续LBL    3LD     SM0.1MOVW   3, VW198           // 步骤=3(RTC正常)
// BCD转秒 - RTC(VD_RTC_Now_Sec)MOVR   0.0, VD186         // 清VD_RTC_Now_SecBTI    VB903, AC0         // BCD→INT(时)ITD    AC0, AC0           // INT→DINTDTR    AC0, AC0           // DINT→REAL*R     3600.0, AC0        // ×3600+R     AC0, VD186         // 累加到VD_RTC_Now_SecBTI    VB904, AC0         // 分ITD    AC0, AC0DTR    AC0, AC0*R     60.0, AC0+R     AC0, VD186BTI    VB905, AC0         // 秒ITD    AC0, AC0DTR    AC0, AC0+R     AC0, VD186
// BCD转秒 - DT10(VD_DT10_Sec)MOVR   0.0, VD190         // 清VD_DT10_SecBTI    VB13, AC0          // DT10时ITD    AC0, AC0DTR    AC0, AC0*R     3600.0, AC0+R     AC0, VD190BTI    VB14, AC0          // 分ITD    AC0, AC0DTR    AC0, AC0*R     60.0, AC0+R     AC0, VD190BTI    VB15, AC0          // 秒ITD    AC0, AC0DTR    AC0, AC0+R     AC0, VD190MOVW   4, VW198           // 步骤=4(BCD转秒完成)
// VD_S5_Elapsed重算(仅保持S5且下缸=满时)LD     V1.7               // 下缸=满AW=    VW2, 6             // 且状态机=S5MOVR   VD186, VD178       // 满足:VD_S5_Elapsed = RTC秒-R     VD190, VD178       // - DT10秒 = 断电期间经过秒数MOVW   5, VW198           // 步骤=5(Elapsed重算完成)JMP    5                  // → 状态恢复
// 下缸=空 或 非S5 时VD_S5_Elapsed=0LD     SM0.0MOVR   0.0, VD178         // Elapsed=0MOVW   5, VW198
// ===== 状态机恢复策略 =====LBL    5LDW=   VW2, 0JMP    6                  // S0保持
// S5保持(断电续跑) —— 【2026-09-29修复】加前提://   仅当下缸=满(实验确实在跑,V1.7=1)或上缸有配液任务(VW418≠0)时才续跑;//   否则判定为断电残留死状态(典型现象: 上电后上缸空闲+下缸显示S5空等,//   停止/启动都脱不了困,只能断电复位), 清状态回S0(复用LBL 10清理段)。// 用V60.2/V60.3草稿位缓存条件,避免LDW+V1.7/OLD栈混叠。LDW=   VW2, 6=      V60.2              // V60.2=断电时处于S5LD     V1.7               // 下缸=满LDW<>  VW418, 0           // 或上缸子流程有任务OLD=      V60.3              // V60.3=S5续跑前提成立LD     V60.2A      V60.3JMP    6                  // 前提满足 → S5保持(断电续跑)LD     V60.2AN     V60.3JMP    10                 // 无前提 → 残留死状态,复用S_ERROR回S0清理段(LBL 10)
LDW=   VW2, 8JMP    6                  // S7保持(锁定态)
// S_ERROR: 无实际故障则转S0，否则保持LDW=   VW2, 99JMP    7
// S1~S6: 阀门/泵动作中断 → 转S_ERRORLD     SM0.0MOVB   0, QB0             // 阀门关/泵停/NC电磁阀失电(安全)MOVW   99, VW2            // 转S_ERRORS      V300.4, 1          // 置急停锁存(需人工复位)// ★ 2026-09-14新增: 清运行中间状态,防止断电恢复后带半拉子S1状态运行R      V1.0, 1            // 清启动握手位R      M10.2, 1           // 清S1首次进入标志 【2026-09-29新增】FILL   0, VW260, 8        // 清 VB260~VB275 (阀A/B/C诊断子状态)R      T50, 6             // 清 T50~T55 (阀A/B诊断计时器)MOVW   7, VW198           // 步骤=7(状态机转S_ERROR)
// S_ERROR特殊处理LBL    7LD     V300.4             // 急停锁存O      V300.5             // 或继电器故障O      I1.1               // 或急停触发LDW<>  VW6, 0             // 或有活动报警OLDJMP    6                  // 任一满足 → 保持S_ERROR
// 无实际故障 → 转S0// 【2026-09-29】本段同时是S5残留死状态的清理落点(S5无续跑前提时JMP 10),//   复用同一段清理指令,不为S5单写副本(省程序存储器,ST20仅剩12KB余量紧张)LBL    10LD     SM0.1MOVB   0, QB0             // 输出安全状态R      Q0.7, 1            // 清报警声音MOVW   0, VW2             // 转S0// ★ 2026-09-14新增: 从S_ERROR回S0时同样清理残留状态R      V1.0, 1            // 清启动握手位R      M10.2, 1           // 清S1首次进入标志 【2026-09-29新增】FILL   0, VW260, 8        // 清 VB260~VB275 (阀A/B/C诊断子状态)R      T50, 6             // 清 T50~T55 (阀A/B诊断计时器)// 【v2.2 新增】断电恢复时清理上缸子流程 + 双倒计时器MOVW   0, VW418                     // 上缸配液子流程状态清零MOVW   0, VW400                     // 换水计数清零(防御性) 【v2.3.2迁移: 原VW306与手动命令位V306.0~V307.3重叠】R      M16.0, 4                     // M16.0~M16.3 连续清零R      T63, 1                       // [已修复 v2.2] 清 1s 脉冲定时器R      T49, 1                       // 清 S4 转移计时器MOVR   0.0, VD248                   // [已修复 v2.2] 清 TimerA_ElapsedMOVR   0.0, VD252                   // [已修复 v2.2] 清 TimerB_ElapsedMOVR   0.0, VD256                   // 清 TimerA 显示值MOVR   0.0, VD244                   // 清 TimerB 显示值MOVW   6, VW198           // 步骤=6(状态恢复完成)
// 保持原状态LBL    6MOVW   6, VW198           // 步骤=6(状态恢复完成)// SBR 自然结束,返回到 FC0 的 LBL 2 (S M16.4,1)

// ============================================================// 文件结束// ============================================================

BTI    VB14, AC0
ITD    AC0, AC0
DTR    AC0, AC0
*R     60.0, AC0
+R     AC0, VD190
BTI    VB15, AC0
ITD    AC0, AC0
DTR    AC0, AC0
+R     AC0, VD190
MOVW   4, VW198
LD     V1.7
AW=    VW2, 6
MOVR   VD186, VD178
-R     VD190, VD178
MOVW   5, VW198
JMP    5
LD     SM0.0
MOVR   0.0, VD178
MOVW   5, VW198
LBL    5
LDW=   VW2, 0
JMP    6
LDW=   VW2, 6
=      V60.2
LD     V1.7
LDW<>  VW418, 0
OLD
=      V60.3
LD     V60.2
A      V60.3
JMP    6
LD     V60.2
AN     V60.3
JMP    10
LDW=   VW2, 8
JMP    6
LDW=   VW2, 99
JMP    7
LD     SM0.0
MOVB   0, QB0
MOVW   99, VW2
S      V300.4, 1
R      V1.0, 1
R      M10.2, 1
FILL   0, VW260, 8
R      T50, 6
MOVW   7, VW198
LBL    7
LD     V300.4
O      V300.5
O      I1.1
LDW<>  VW6, 0
OLD
JMP    6
LBL    10
LD     SM0.1
MOVB   0, QB0
R      Q0.7, 1
MOVW   0, VW2
R      V1.0, 1
R      M10.2, 1
FILL   0, VW260, 8
R      T50, 6
MOVW   0, VW418
MOVW   0, VW400
R      M16.0, 4
R      T63, 1
R      T49, 1
MOVR   0.0, VD248
MOVR   0.0, VD252
MOVR   0.0, VD256
MOVR   0.0, VD244
MOVW   6, VW198
LBL    6
MOVW   6, VW198
END_SUBROUTINE_BLOCK
SUBROUTINE_BLOCK PumpErrExit:SBR27
TITLE=// ============================================================
// // 文件: FC13A_PumpErrExit.stl
// // 功能: FC13 公共泵错误退出处理(停泵+转S_ERROR+清握手)
// // Story: 压缩 FC13 程序体积,提取 NETWORK 2/4/7/10/13 重复的错误退出代码
// // 说明: 本 FC 由 FC13 各错误路径 CALL 调用,统一执行:
// //       1. 安全停潜水泵 Q0.0/Q0.1
// //       2. 置位注射泵报警位 V303.4
// //       3. 状态机转 S_ERROR(VW2=99)
// //       4. 清 S3 子状态 VW226=0
// //       5. 清写握手位 M12.0/M11.6/M11.7
// //       6. 清运动标志 M12.1/M12.2
// //       7. 清超时定时器 T102
// // 调用方: FC13 NETWORK 2(全局错误检测) / NETWORK 4(子状态1/5写失败)
// //         NETWORK 7(子状态3/7写失败)
// // ============================================================
BEGIN
Network 1
//  FC13泵错误退出公共处理
//  由FC13各错误路径CALL,统一执行安全停泵+转S_ERROR+清握手
R      Q0.0, 1                     // 停潜水泵1
R      Q0.1, 1                       // 停潜水泵2S      V303.4, 1                     // 确保报警位MOVW   99, VW2                       // 转S_ERRORMOVW   0, VW226                      // 清子状态R      M12.0, 1                      // 清写完成R      M12.1, 1                      // 清抽液运动标志R      M12.2, 1                      // 清排液运动标志R      M11.6, 1                      // 清写请求R      M11.7, 1                      // 清写忙R      T102, 1                       // 清超时定时器

// ============================================================// 文件结束// 说明://   1. 本 FC 仅在错误路径被 CALL 调用,不单独从 OB1 调用//   2. 调用前由调用方保证执行条件(已检测到 V303.4 或 VW4≥4)//   3. 所有复位操作为幂等,重复调用安全// ============================================================

END_SUBROUTINE_BLOCK
SUBROUTINE_BLOCK AlarmReset_Common:SBR28
TITLE=// ============================================================
// // 文件: FC3A_AlarmReset_Common.stl
// // 功能: FC3 公共报警位复位逻辑（条件消失则复位）
// // Story: 压缩 FC3 程序体积，提取 NETWORK 4/5 重复代码
// // 说明: 本 FC 仅包含一般故障级报警位的条件消失自动复位逻辑，
// //       漫溢级(V300.0~3)、急停(V300.4)、继电器故障(V300.5)、
// //       节奏滞后(V300.6/7)不由本 FC 处理。
// //       V303.6(单轮换水周期超时)也由 FC3 NETWORK 4 (V0.3上升沿) 单独复位(2026-09-25):
// //       FC40注4要求必须人工确认,不受V200.0自动模式影响,放入本FC会被
// //       NETWORK 5(自动恢复)每扫描调用而自动清除,故刻意排除。
// //       注意: FC3复位时同步清零VD248/VD252,否则NET6同扫描重报(死锁)
// // 调用方: FC3 NETWORK 4(人工确认时)、FC3 NETWORK 5(自动恢复模式)
// // ============================================================
//
BEGIN
Network 1
//  阀A类：条件消失则复位
LD     V301.0                      // 阀A关后仍有流
AN     I0.0                          // 流量开关A已OFF
R      V301.0, 1

LD     V301.2                        // 阀A关到位超时
A      I8.1                          // 阀A关到位反馈已ON
R      V301.2, 1

LD     V301.3                        // 阀A关到位但仍有流
AN     I0.0                          // 流量开关A已OFF
R      V301.3, 1

LD     V301.4                        // 阀A开到位超时
A      I8.0                          // 阀A开到位反馈已ON
R      V301.4, 1

LD     V301.5                        // 阀A开到位但无流
A      I0.0                          // 流量开关A已ON
R      V301.5, 1

LD     V301.6                        // S5触发S1时上缸≠空
AN     V1.6                          // 上缸已=空
R      V301.6, 1


// 阀B/C类：条件消失则复位
LD     V302.0                        // 阀B诊断异常
LD     I0.1                          // 流量开关B=ON
O      I0.6                          // 或液位计A-低位=ON
ALD
R      V302.0, 1

LD     V302.1                        // 阀B开到位超时
A      I8.2
R      V302.1, 1

LD     V302.2                        // 阀B开到位但无流
A      I0.1
R      V302.2, 1

LD     V302.3                        // 阀B关到位超时
A      I8.3
R      V302.3, 1

LD     V302.4                        // 阀B关到位但仍有流
AN     I0.1
R      V302.4, 1

// 【v10.4硬件变更】V302.5(报警码45)/V302.7(报警码47)已废弃为保留位,
//   FC32不再置位,此处删除原基于I0.2的复位条件
LD     V302.6                        // 阀C开到位超时
A      I8.4
R      V302.6, 1


// 其他类：条件消失则复位
// 注: V303.0(报警码60)现覆盖关到位超时+排水超时两种触发,
//     复位条件统一为阀C关到位反馈I8.5=ON
LD     V303.0                        // 阀C关到位超时/排水超时
A      I8.5
R      V303.0, 1

// 【v10.4硬件变更】V303.1(报警码61,阀C关到位仍有流)已废弃为保留位,
//   内漏判定依赖I0.2已去除,此处删除原复位条件
LD     V303.4                        // 注射泵通讯异常
AW=    VW4, 0                        // 状态码=0(空闲正常)
R      V303.4, 1

// 注: V303.5(RTC丢失)不自动清除，需HMI校时后确认


// ============================================================
// 文件结束
// 说明:
//   1. 本 FC 被 FC3 调用，不要单独从 OB1 调用
//   2. 调用前由调用方保证执行时机（NETWORK 4 的 V0.3 上升沿 / NETWORK 5 的自动模式）
//   3. 报警位复位后，下一周期 FC3 NETWORK 1 会重算 VW6
// ============================================================

END_SUBROUTINE_BLOCK
INTERRUPT_BLOCK MBUSM2:INT0
TITLE=This code is property of Siemens Industry, Inc.
BEGIN
Network 1 // 此 POU 针对编辑和查看设置了密码保护.

END_INTERRUPT_BLOCK
